PROGRAM EM06_Robot
VAR
END_VAR

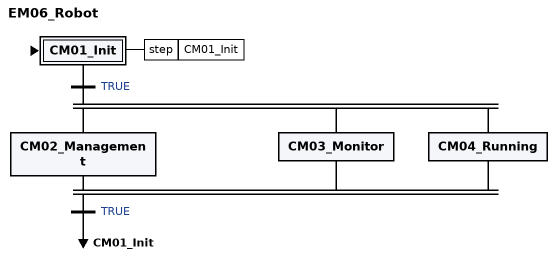
INITIAL_STEP CM01_Init:
    CM01_Init(N);  // step action
END_STEP
TRANSITION FROM CM01_Init TO (CM02_Management, CM03_Monitor, CM04_Running)
    := TRUE;
END_TRANSITION
STEP CM02_Management:
END_STEP
STEP CM03_Monitor:
END_STEP
STEP CM04_Running:
END_STEP
TRANSITION FROM (CM02_Management, CM03_Monitor, CM04_Running) TO CM01_Init
    := TRUE;
END_TRANSITION

ACTION CM01_Init:

END_ACTION

ACTION CM02_Management:
// NETWORK 1
END_ACTION

ACTION CM03_Monitor:
// NETWORK 1
END_ACTION

ACTION CM04_Running:
// NETWORK 1
END_ACTION

END_PROGRAM

(* stored: Version 1.1.0.1, ProductVersion 3.1.4024.9
   POU EM06_Robot: Id {bf31a6a4-6cb3-4143-b13c-4e3d1a94a9b3}, SpecialFunc None
   Action CM01_Init: Id {942e7d26-266d-4710-bc8a-4c4383a26528}
   Action CM02_Management: Id {d99a6982-1287-4a71-8522-f2e3b9427739}
   Action CM03_Monitor: Id {5c81fae1-d47c-423b-930f-cb85f7348b34}
   Action CM04_Running: Id {b9beb71e-7f36-42f1-9a58-50f44cc39b0b} *)
